ABB RobotStudio station: FinalProject.rsstnx

Station FinalProject (saved by RobotStudio 24.4.11080.0)
Controller IRB140_6_81
  mechanical unit ROB_1: IRB140_6_81_C_03, 6 joints, base frame (0, 0, 0) mm
Layout (positions relative to the parent item):
  - IRB140_6_81_C_03 [mechanism, from %ABB.RobotStudio.Models.IRB140%\IRB140_6_81_C_G_03.rslib] at (0, 0, 0) mm; joint values [0, 0, 0, 0, 0, 0] (rad or m)
  - VacuumGripper [mechanism] at (515, 0, 712) mm, rotated rx 0 ry 90 rz 0 deg
      TCP VacuumGripper at (122.78, 0, 0) mm, rotated rx 90 ry 45 rz 90 deg
      links: FakeEE
Attachment: VacuumGripper is attached to IRB140_6_81_C_03 / Link6
Targets, tools, work objects and paths stored in the station, written as RAPID:
! task T_ROB1
MODULE Numbers
  CONST robtarget T_01:=[[-310.742,318.894,0],[1,0,0,0],[0,0,0,0],[9E+09,9E+09,9E+09,9E+09,9E+09,9E+09]];
  CONST robtarget T_02:=[[-285.702,367.273,0],[1,0,0,0],[0,-1,0,0],[9E+09,9E+09,9E+09,9E+09,9E+09,9E+09]];
  CONST robtarget T_03:=[[-206.529,382.913,0],[1,0,0,0],[0,-1,0,0],[9E+09,9E+09,9E+09,9E+09,9E+09,9E+09]];
  CONST robtarget T_04:=[[-128.165,367.435,0],[1,0,0,0],[0,-2,1,0],[9E+09,9E+09,9E+09,9E+09,9E+09,9E+09]];
  CONST robtarget T_05:=[[-102.477,318.894,0],[1,0,0,0],[-2,0,1,6],[9E+09,9E+09,9E+09,9E+09,9E+09,9E+09]];
  CONST robtarget T_06:=[[-127.679,270.676,0],[1,0,0,0],[-2,0,1,6],[9E+09,9E+09,9E+09,9E+09,9E+09,9E+09]];
  CONST robtarget T_07:=[[-206.691,255.036,0],[1,0,0,0],[-1,0,-1,0],[9E+09,9E+09,9E+09,9E+09,9E+09,9E+09]];
  CONST robtarget T_08:=[[-284.811,270.514,0],[1,0,0,0],[-1,0,-1,0],[9E+09,9E+09,9E+09,9E+09,9E+09,9E+09]];
  CONST robtarget T_09:=[[-310.742,318.894,0],[1,0,0,0],[0,-1,0,0],[9E+09,9E+09,9E+09,9E+09,9E+09,9E+09]];
  CONST robtarget T_11:=[[-106.691,366.707,0],[1,0,0,0],[0,0,-1,1],[9E+09,9E+09,9E+09,9E+09,9E+09,9E+09]];
  CONST robtarget T_12:=[[-106.691,269.138,0],[1,0,0,0],[0,0,-1,1],[9E+09,9E+09,9E+09,9E+09,9E+09,9E+09]];
  CONST robtarget T_13:=[[-106.691,317.923,0],[1,0,0,0],[0,0,-1,1],[9E+09,9E+09,9E+09,9E+09,9E+09,9E+09]];
  CONST robtarget T_14:=[[-307.339,315.005,0],[1,0,0,0],[0,0,-1,1],[9E+09,9E+09,9E+09,9E+09,9E+09,9E+09]];
  CONST robtarget T_15:=[[-285.297,336.399,0],[1,0,0,0],[0,1,-2,1],[9E+09,9E+09,9E+09,9E+09,9E+09,9E+09]];
  CONST robtarget T_16:=[[-279.462,366.707,0],[1,0,0,0],[0,1,-2,1],[9E+09,9E+09,9E+09,9E+09,9E+09,9E+09]];
  CONST robtarget T_21:=[[-106.691,261.009,0],[1,0,0,0],[0,-1,0,0],[9E+09,9E+09,9E+09,9E+09,9E+09,9E+09]];
  CONST robtarget T_22:=[[-106.691,384.347,0],[1,0,0,0],[0,-2,1,0],[9E+09,9E+09,9E+09,9E+09,9E+09,9E+09]];
  CONST robtarget T_23:=[[-129.867,359.226,0],[1,0,0,0],[0,-2,1,0],[9E+09,9E+09,9E+09,9E+09,9E+09,9E+09]];
  CONST robtarget T_24:=[[-153.206,334.509,0],[1,0,0,0],[0,-2,1,0],[9E+09,9E+09,9E+09,9E+09,9E+09,9E+09]];
  CONST robtarget T_25:=[[-181.731,306.39,0],[1,0,0,0],[0,-1,0,0],[9E+09,9E+09,9E+09,9E+09,9E+09,9E+09]];
  CONST robtarget T_26:=[[-215.929,279.647,0],[1,0,0,0],[0,-1,0,0],[9E+09,9E+09,9E+09,9E+09,9E+09,9E+09]];
  CONST robtarget T_27:=[[-255.961,269.274,0],[1,0,0,0],[0,-1,0,0],[9E+09,9E+09,9E+09,9E+09,9E+09,9E+09]];
  CONST robtarget T_28:=[[-296.075,285.077,0],[1,0,0,0],[0,-1,0,0],[9E+09,9E+09,9E+09,9E+09,9E+09,9E+09]];
  CONST robtarget T_29:=[[-310.905,328.918,0],[1,0,0,0],[0,-1,0,0],[9E+09,9E+09,9E+09,9E+09,9E+09,9E+09]];
  CONST robtarget T_210:=[[-306.934,357.038,0],[1,0,0,0],[0,-1,0,0],[9E+09,9E+09,9E+09,9E+09,9E+09,9E+09]];
  CONST robtarget T_211:=[[-298.911,380.133,0],[1,0,0,0],[0,-1,0,0],[9E+09,9E+09,9E+09,9E+09,9E+09,9E+09]];
  CONST robtarget T_31:=[[-298.587,375.377,0],[1,0,0,0],[0,-1,0,0],[9E+09,9E+09,9E+09,9E+09,9E+09,9E+09]];
  CONST robtarget T_32:=[[-307.096,351.633,0],[1,0,0,0],[0,-1,0,0],[9E+09,9E+09,9E+09,9E+09,9E+09,9E+09]];
  CONST robtarget T_33:=[[-310.905,323.189,0],[1,0,0,0],[0,-1,0,0],[9E+09,9E+09,9E+09,9E+09,9E+09,9E+09]];
  CONST robtarget T_34:=[[-308.149,299.445,0],[1,0,0,0],[0,-1,0,0],[9E+09,9E+09,9E+09,9E+09,9E+09,9E+09]];
  CONST robtarget T_35:=[[-299.559,281.049,0],[1,0,0,0],[0,-1,0,0],[9E+09,9E+09,9E+09,9E+09,9E+09,9E+09]];
  CONST robtarget T_36:=[[-284.081,267.759,0],[1,0,0,0],[0,-1,0,0],[9E+09,9E+09,9E+09,9E+09,9E+09,9E+09]];
  CONST robtarget T_37:=[[-262.606,263.221,0],[1,0,0,0],[0,-1,0,0],[9E+09,9E+09,9E+09,9E+09,9E+09,9E+09]];
  CONST robtarget T_38:=[[-233.595,274.08,0],[1,0,0,0],[0,-1,0,0],[9E+09,9E+09,9E+09,9E+09,9E+09,9E+09]];
  CONST robtarget T_39:=[[-217.874,300.174,0],[1,0,0,0],[0,-1,0,0],[9E+09,9E+09,9E+09,9E+09,9E+09,9E+09]];
  CONST robtarget T_310:=[[-215.199,340.044,0],[1,0,0,0],[0,-1,0,0],[9E+09,9E+09,9E+09,9E+09,9E+09,9E+09]];
  CONST robtarget T_311:=[[-215.929,300.174,0],[1,0,0,0],[0,-1,0,0],[9E+09,9E+09,9E+09,9E+09,9E+09,9E+09]];
  CONST robtarget T_312:=[[-202.963,273.27,0],[1,0,0,0],[0,-1,0,0],[9E+09,9E+09,9E+09,9E+09,9E+09,9E+09]];
  CONST robtarget T_313:=[[-188.214,263.221,0],[1,0,0,0],[0,-1,0,0],[9E+09,9E+09,9E+09,9E+09,9E+09,9E+09]];
  CONST robtarget T_314:=[[-166.01,259.331,0],[1,0,0,0],[0,-1,0,0],[9E+09,9E+09,9E+09,9E+09,9E+09,9E+09]];
  CONST robtarget T_315:=[[-141.131,263.95,0],[1,0,0,0],[0,-1,0,0],[9E+09,9E+09,9E+09,9E+09,9E+09,9E+09]];
  CONST robtarget T_316:=[[-120.953,276.997,0],[1,0,0,0],[0,-1,0,0],[9E+09,9E+09,9E+09,9E+09,9E+09,9E+09]];
  CONST robtarget T_317:=[[-107.177,298.148,0],[1,0,0,0],[0,-2,1,0],[9E+09,9E+09,9E+09,9E+09,9E+09,9E+09]];
  CONST robtarget T_318:=[[-102.477,326.268,0],[1,0,0,0],[0,-2,1,0],[9E+09,9E+09,9E+09,9E+09,9E+09,9E+09]];
  CONST robtarget T_319:=[[-106.123,356.09,0],[1,0,0,0],[0,-2,1,0],[9E+09,9E+09,9E+09,9E+09,9E+09,9E+09]];
  CONST robtarget T_320:=[[-114.794,380.887,0],[1,0,0,0],[0,-2,1,0],[9E+09,9E+09,9E+09,9E+09,9E+09,9E+09]];
  CONST robtarget T_41:=[[-106.691,281.323,0],[1,0,0,0],[-1,-1,0,1],[9E+09,9E+09,9E+09,9E+09,9E+09,9E+09]];
  CONST robtarget T_42:=[[-306.691,281.323,0],[1,0,0,0],[0,0,-1,1],[9E+09,9E+09,9E+09,9E+09,9E+09,9E+09]];
  CONST robtarget T_43:=[[-306.691,305.958,0],[1,0,0,0],[0,1,-2,1],[9E+09,9E+09,9E+09,9E+09,9E+09,9E+09]];
  CONST robtarget T_44:=[[-203.611,395.424,0],[1,0,0,0],[0,1,-2,1],[9E+09,9E+09,9E+09,9E+09,9E+09,9E+09]];
  CONST robtarget T_45:=[[-175.41,395.424,0],[1,0,0,0],[0,1,-2,1],[9E+09,9E+09,9E+09,9E+09,9E+09,9E+09]];
  CONST robtarget T_46:=[[-175.41,257.498,0],[1,0,0,0],[0,1,-2,1],[9E+09,9E+09,9E+09,9E+09,9E+09,9E+09]];
  CONST robtarget T_51:=[[-306.691,269.007,0],[1,0,0,0],[0,1,-2,1],[9E+09,9E+09,9E+09,9E+09,9E+09,9E+09]];
  CONST robtarget T_52:=[[-306.691,378.732,0],[1,0,0,0],[0,1,-2,1],[9E+09,9E+09,9E+09,9E+09,9E+09,9E+09]];
  CONST robtarget T_53:=[[-223.611,378.732,0],[1,0,0,0],[0,1,-2,1],[9E+09,9E+09,9E+09,9E+09,9E+09,9E+09]];
  CONST robtarget T_54:=[[-229.867,352.962,0],[1,0,0,0],[0,1,-2,1],[9E+09,9E+09,9E+09,9E+09,9E+09,9E+09]];
  CONST robtarget T_55:=[[-231.002,334.809,0],[1,0,0,0],[0,1,-2,1],[9E+09,9E+09,9E+09,9E+09,9E+09,9E+09]];
  CONST robtarget T_56:=[[-228.49,308.796,0],[1,0,0,0],[0,1,-2,1],[9E+09,9E+09,9E+09,9E+09,9E+09,9E+09]];
  CONST robtarget T_57:=[[-218.522,288.456,0],[1,0,0,0],[0,1,-2,1],[9E+09,9E+09,9E+09,9E+09,9E+09,9E+09]];
  CONST robtarget T_58:=[[-199.721,273.221,0],[1,0,0,0],[0,1,-2,1],[9E+09,9E+09,9E+09,9E+09,9E+09,9E+09]];
  CONST robtarget T_59:=[[-170.224,267.873,0],[1,0,0,0],[0,1,-2,1],[9E+09,9E+09,9E+09,9E+09,9E+09,9E+09]];
  CONST robtarget T_510:=[[-143.482,272.492,0],[1,0,0,0],[0,0,-1,1],[9E+09,9E+09,9E+09,9E+09,9E+09,9E+09]];
  CONST robtarget T_511:=[[-122.088,285.539,0],[1,0,0,0],[0,0,-1,1],[9E+09,9E+09,9E+09,9E+09,9E+09,9E+09]];
  CONST robtarget T_512:=[[-107.744,306.527,0],[1,0,0,0],[0,0,-1,1],[9E+09,9E+09,9E+09,9E+09,9E+09,9E+09]];
  CONST robtarget T_513:=[[-102.477,334.647,0],[1,0,0,0],[0,0,-1,1],[9E+09,9E+09,9E+09,9E+09,9E+09,9E+09]];
  CONST robtarget T_514:=[[-105.637,362.848,0],[1,0,0,0],[0,0,-1,1],[9E+09,9E+09,9E+09,9E+09,9E+09,9E+09]];
  CONST robtarget T_515:=[[-113.822,386.997,0],[1,0,0,0],[0,0,-1,1],[9E+09,9E+09,9E+09,9E+09,9E+09,9E+09]];
  CONST robtarget T_61:=[[-307.663,280.947,0],[1,0,0,0],[0,0,-1,1],[9E+09,9E+09,9E+09,9E+09,9E+09,9E+09]];
  CONST robtarget T_62:=[[-310.418,303.638,0],[1,0,0,0],[0,1,-2,1],[9E+09,9E+09,9E+09,9E+09,9E+09,9E+09]];
  CONST robtarget T_63:=[[-301.909,343.346,0],[1,0,0,0],[0,1,-2,1],[9E+09,9E+09,9E+09,9E+09,9E+09,9E+09]];
  CONST robtarget T_64:=[[-278.165,371.385,0],[1,0,0,0],[0,1,-2,1],[9E+09,9E+09,9E+09,9E+09,9E+09,9E+09]];
  CONST robtarget T_65:=[[-241.618,387.916,0],[1,0,0,0],[0,1,-2,1],[9E+09,9E+09,9E+09,9E+09,9E+09,9E+09]];
  CONST robtarget T_66:=[[-194.535,393.265,0],[1,0,0,0],[0,1,-2,1],[9E+09,9E+09,9E+09,9E+09,9E+09,9E+09]];
  CONST robtarget T_67:=[[-149.721,387.43,0],[1,0,0,0],[0,1,-2,1],[9E+09,9E+09,9E+09,9E+09,9E+09,9E+09]];
  CONST robtarget T_68:=[[-120.629,371.223,0],[1,0,0,0],[0,0,-1,1],[9E+09,9E+09,9E+09,9E+09,9E+09,9E+09]];
  CONST robtarget T_69:=[[-107.015,351.693,0],[1,0,0,0],[0,0,-1,1],[9E+09,9E+09,9E+09,9E+09,9E+09,9E+09]];
  CONST robtarget T_610:=[[-102.477,327.138,0],[1,0,0,0],[0,0,-1,1],[9E+09,9E+09,9E+09,9E+09,9E+09,9E+09]];
  CONST robtarget T_611:=[[-107.258,302.503,0],[1,0,0,0],[0,0,-1,1],[9E+09,9E+09,9E+09,9E+09,9E+09,9E+09]];
  CONST robtarget T_612:=[[-121.277,282.406,0],[1,0,0,0],[0,0,-1,1],[9E+09,9E+09,9E+09,9E+09,9E+09,9E+09]];
  CONST robtarget T_613:=[[-143.076,268.71,0],[1,0,0,0],[0,0,-1,1],[9E+09,9E+09,9E+09,9E+09,9E+09,9E+09]];
  CONST robtarget T_614:=[[-171.52,263.605,0],[1,0,0,0],[0,1,-2,1],[9E+09,9E+09,9E+09,9E+09,9E+09,9E+09]];
  CONST robtarget T_615:=[[-201.504,268.954,0],[1,0,0,0],[0,1,-2,1],[9E+09,9E+09,9E+09,9E+09,9E+09,9E+09]];
  CONST robtarget T_616:=[[-222.574,285.323,0],[1,0,0,0],[0,1,-2,1],[9E+09,9E+09,9E+09,9E+09,9E+09,9E+09]];
  CONST robtarget T_617:=[[-232.055,303.638,0],[1,0,0,0],[0,1,-2,1],[9E+09,9E+09,9E+09,9E+09,9E+09,9E+09]];
  CONST robtarget T_618:=[[-234.405,324.059,0],[1,0,0,0],[0,1,-2,1],[9E+09,9E+09,9E+09,9E+09,9E+09,9E+09]];
  CONST robtarget T_619:=[[-230.759,346.101,0],[1,0,0,0],[0,1,-2,1],[9E+09,9E+09,9E+09,9E+09,9E+09,9E+09]];
  CONST robtarget T_620:=[[-220.467,365.712,0],[1,0,0,0],[0,1,-2,1],[9E+09,9E+09,9E+09,9E+09,9E+09,9E+09]];
  CONST robtarget T_621:=[[-194.535,393.265,0],[1,0,0,0],[0,1,-2,1],[9E+09,9E+09,9E+09,9E+09,9E+09,9E+09]];
  CONST robtarget T_71:=[[-306.691,388.239,0],[1,0,0,0],[0,-1,0,0],[9E+09,9E+09,9E+09,9E+09,9E+09,9E+09]];
  CONST robtarget T_72:=[[-306.691,261.334,0],[1,0,0,0],[0,-1,0,0],[9E+09,9E+09,9E+09,9E+09,9E+09,9E+09]];
  CONST robtarget T_73:=[[-106.691,347.882,0],[1,0,0,0],[0,-1,0,0],[9E+09,9E+09,9E+09,9E+09,9E+09,9E+09]];
  CONST robtarget T_81:=[[-214.308,359.688,0],[1,0,0,0],[0,1,-2,1],[9E+09,9E+09,9E+09,9E+09,9E+09,9E+09]];
  CONST robtarget T_82:=[[-233.109,381.568,0],[1,0,0,0],[0,1,-2,1],[9E+09,9E+09,9E+09,9E+09,9E+09,9E+09]];
  CONST robtarget T_83:=[[-258.554,388.699,0],[1,0,0,0],[0,1,-2,1],[9E+09,9E+09,9E+09,9E+09,9E+09,9E+09]];
  CONST robtarget T_84:=[[-296.156,371.681,0],[1,0,0,0],[0,1,-2,1],[9E+09,9E+09,9E+09,9E+09,9E+09,9E+09]];
  CONST robtarget T_85:=[[-311.229,328.407,0],[1,0,0,0],[0,1,-2,1],[9E+09,9E+09,9E+09,9E+09,9E+09,9E+09]];
  CONST robtarget T_86:=[[-296.966,284.728,0],[1,0,0,0],[0,1,-2,1],[9E+09,9E+09,9E+09,9E+09,9E+09,9E+09]];
  CONST robtarget T_87:=[[-260.337,268.278,0],[1,0,0,0],[0,1,-2,1],[9E+09,9E+09,9E+09,9E+09,9E+09,9E+09]];
  CONST robtarget T_88:=[[-233.757,276.138,0],[1,0,0,0],[0,1,-2,1],[9E+09,9E+09,9E+09,9E+09,9E+09,9E+09]];
  CONST robtarget T_89:=[[-213.174,298.748,0],[1,0,0,0],[0,1,-2,1],[9E+09,9E+09,9E+09,9E+09,9E+09,9E+09]];
  CONST robtarget T_810:=[[-213.498,359.688,0],[1,0,0,0],[0,1,-2,1],[9E+09,9E+09,9E+09,9E+09,9E+09,9E+09]];
  CONST robtarget T_811:=[[-191.78,384.89,0],[1,0,0,0],[0,1,-2,1],[9E+09,9E+09,9E+09,9E+09,9E+09,9E+09]];
  CONST robtarget T_812:=[[-161.958,393.561,0],[1,0,0,0],[0,1,-2,1],[9E+09,9E+09,9E+09,9E+09,9E+09,9E+09]];
  CONST robtarget T_813:=[[-138.457,389.185,0],[1,0,0,0],[0,0,-1,1],[9E+09,9E+09,9E+09,9E+09,9E+09,9E+09]];
  CONST robtarget T_814:=[[-119.332,376.381,0],[1,0,0,0],[0,0,-1,1],[9E+09,9E+09,9E+09,9E+09,9E+09,9E+09]];
  CONST robtarget T_815:=[[-106.61,355.555,0],[1,0,0,0],[0,0,-1,1],[9E+09,9E+09,9E+09,9E+09,9E+09,9E+09]];
  CONST robtarget T_816:=[[-102.152,328.407,0],[1,0,0,0],[0,0,-1,1],[9E+09,9E+09,9E+09,9E+09,9E+09,9E+09]];
  CONST robtarget T_817:=[[-119.494,281.892,0],[1,0,0,0],[0,0,-1,1],[9E+09,9E+09,9E+09,9E+09,9E+09,9E+09]];
  CONST robtarget T_818:=[[-162.444,263.253,0],[1,0,0,0],[0,1,-2,1],[9E+09,9E+09,9E+09,9E+09,9E+09,9E+09]];
  CONST robtarget T_819:=[[-192.59,272.249,0],[1,0,0,0],[0,1,-2,1],[9E+09,9E+09,9E+09,9E+09,9E+09,9E+09]];
  CONST robtarget T_820:=[[-212.363,298.748,0],[1,0,0,0],[0,1,-2,1],[9E+09,9E+09,9E+09,9E+09,9E+09,9E+09]];
  CONST robtarget T_821:=[[-214.308,359.688,0],[1,0,0,0],[0,1,-2,1],[9E+09,9E+09,9E+09,9E+09,9E+09,9E+09]];
  CONST robtarget T_91:=[[-105.556,371.949,0],[1,0,0,0],[0,0,-1,1],[9E+09,9E+09,9E+09,9E+09,9E+09,9E+09]];
  CONST robtarget T_92:=[[-102.801,349.258,0],[1,0,0,0],[0,0,-1,1],[9E+09,9E+09,9E+09,9E+09,9E+09,9E+09]];
  CONST robtarget T_93:=[[-110.986,309.388,0],[1,0,0,0],[0,0,-1,1],[9E+09,9E+09,9E+09,9E+09,9E+09,9E+09]];
  CONST robtarget T_94:=[[-134.729,281.673,0],[1,0,0,0],[0,0,-1,1],[9E+09,9E+09,9E+09,9E+09,9E+09,9E+09]];
  CONST robtarget T_95:=[[-171.682,265.223,0],[1,0,0,0],[0,1,-2,1],[9E+09,9E+09,9E+09,9E+09,9E+09,9E+09]];
  CONST robtarget T_96:=[[-218.684,259.631,0],[1,0,0,0],[0,1,-2,1],[9E+09,9E+09,9E+09,9E+09,9E+09,9E+09]];
  CONST robtarget T_97:=[[-263.903,265.304,0],[1,0,0,0],[0,1,-2,1],[9E+09,9E+09,9E+09,9E+09,9E+09,9E+09]];
  CONST robtarget T_98:=[[-292.752,281.349,0],[1,0,0,0],[0,1,-2,1],[9E+09,9E+09,9E+09,9E+09,9E+09,9E+09]];
  CONST robtarget T_99:=[[-306.123,300.798,0],[1,0,0,0],[0,1,-2,1],[9E+09,9E+09,9E+09,9E+09,9E+09,9E+09]];
  CONST robtarget T_910:=[[-310.742,325.757,0],[1,0,0,0],[0,1,-2,1],[9E+09,9E+09,9E+09,9E+09,9E+09,9E+09]];
  CONST robtarget T_911:=[[-305.799,350.15,0],[1,0,0,0],[0,1,-2,1],[9E+09,9E+09,9E+09,9E+09,9E+09,9E+09]];
  CONST robtarget T_912:=[[-291.942,370.49,0],[1,0,0,0],[0,1,-2,1],[9E+09,9E+09,9E+09,9E+09,9E+09,9E+09]];
  CONST robtarget T_913:=[[-269.9,384.266,0],[1,0,0,0],[0,1,-2,1],[9E+09,9E+09,9E+09,9E+09,9E+09,9E+09]];
  CONST robtarget T_914:=[[-241.699,389.291,0],[1,0,0,0],[0,1,-2,1],[9E+09,9E+09,9E+09,9E+09,9E+09,9E+09]];
  CONST robtarget T_915:=[[-211.472,383.78,0],[1,0,0,0],[0,1,-2,1],[9E+09,9E+09,9E+09,9E+09,9E+09,9E+09]];
  CONST robtarget T_916:=[[-190.645,367.573,0],[1,0,0,0],[0,1,-2,1],[9E+09,9E+09,9E+09,9E+09,9E+09,9E+09]];
  CONST robtarget T_917:=[[-181.245,349.177,0],[1,0,0,0],[0,1,-2,1],[9E+09,9E+09,9E+09,9E+09,9E+09,9E+09]];
  CONST robtarget T_918:=[[-178.814,328.999,0],[1,0,0,0],[0,1,-2,1],[9E+09,9E+09,9E+09,9E+09,9E+09,9E+09]];
  CONST robtarget T_919:=[[-182.136,307.767,0],[1,0,0,0],[0,1,-2,1],[9E+09,9E+09,9E+09,9E+09,9E+09,9E+09]];
  CONST robtarget T_920:=[[-192.752,287.346,0],[1,0,0,0],[0,1,-2,1],[9E+09,9E+09,9E+09,9E+09,9E+09,9E+09]];
  CONST robtarget T_921:=[[-218.684,259.631,0],[1,0,0,0],[0,1,-2,1],[9E+09,9E+09,9E+09,9E+09,9E+09,9E+09]];
  CONST robtarget T_921_2:=[[-218.684,259.631,0],[1,0,0,0],[-1,-2,1,1],[9E+09,9E+09,9E+09,9E+09,9E+09,9E+09]];
  CONST robtarget T_01_2:=[[-310.742,318.894,0],[1,0,0,0],[0,0,0,0],[9E+09,9E+09,9E+09,9E+09,9E+09,9E+09]];
  CONST robtarget T_02_2:=[[-285.702,367.273,0],[1,0,0,0],[-1,0,-1,0],[9E+09,9E+09,9E+09,9E+09,9E+09,9E+09]];
  CONST robtarget T_03_2:=[[-206.529,382.913,0],[1,0,0,0],[-1,0,-1,0],[9E+09,9E+09,9E+09,9E+09,9E+09,9E+09]];
  CONST robtarget T_04_2:=[[-128.165,367.435,0],[1,0,0,0],[-1,0,-1,0],[9E+09,9E+09,9E+09,9E+09,9E+09,9E+09]];
  CONST robtarget T_05_2:=[[-102.477,318.894,0],[1,0,0,0],[-1,0,-1,0],[9E+09,9E+09,9E+09,9E+09,9E+09,9E+09]];
  CONST robtarget T_06_2:=[[-127.679,270.676,0],[1,0,0,0],[-1,1,-2,0],[9E+09,9E+09,9E+09,9E+09,9E+09,9E+09]];
  CONST robtarget T_07_2:=[[-206.691,255.036,0],[1,0,0,0],[-1,0,-1,0],[9E+09,9E+09,9E+09,9E+09,9E+09,9E+09]];
  CONST robtarget T_08_2:=[[-284.811,270.514,0],[1,0,0,0],[-1,0,-1,0],[9E+09,9E+09,9E+09,9E+09,9E+09,9E+09]];
  CONST robtarget T_09_2:=[[-310.742,318.894,0],[1,0,0,0],[-1,0,-1,0],[9E+09,9E+09,9E+09,9E+09,9E+09,9E+09]];
  CONST robtarget T_11_2:=[[-106.691,366.707,0],[1,0,0,0],[-1,1,-2,0],[9E+09,9E+09,9E+09,9E+09,9E+09,9E+09]];
  CONST robtarget T_12_2:=[[-106.691,269.138,0],[1,0,0,0],[-1,1,-2,0],[9E+09,9E+09,9E+09,9E+09,9E+09,9E+09]];
  CONST robtarget T_13_2:=[[-106.691,317.923,0],[1,0,0,0],[-1,1,-2,0],[9E+09,9E+09,9E+09,9E+09,9E+09,9E+09]];
  CONST robtarget T_14_2:=[[-307.339,315.005,0],[1,0,0,0],[-1,1,-2,0],[9E+09,9E+09,9E+09,9E+09,9E+09,9E+09]];
  CONST robtarget T_15_2:=[[-285.297,336.399,0],[1,0,0,0],[-1,0,-1,0],[9E+09,9E+09,9E+09,9E+09,9E+09,9E+09]];
  CONST robtarget T_16_2:=[[-279.462,366.707,0],[1,0,0,0],[-1,0,-1,0],[9E+09,9E+09,9E+09,9E+09,9E+09,9E+09]];
  CONST robtarget T_21_2:=[[-106.691,261.009,0],[1,0,0,0],[-1,1,-2,0],[9E+09,9E+09,9E+09,9E+09,9E+09,9E+09]];
  CONST robtarget T_22_2:=[[-106.691,384.347,0],[1,0,0,0],[-1,1,-2,0],[9E+09,9E+09,9E+09,9E+09,9E+09,9E+09]];
  CONST robtarget T_23_2:=[[-129.867,359.226,0],[1,0,0,0],[-1,1,-2,0],[9E+09,9E+09,9E+09,9E+09,9E+09,9E+09]];
  CONST robtarget T_24_2:=[[-153.206,334.509,0],[1,0,0,0],[-1,0,-1,0],[9E+09,9E+09,9E+09,9E+09,9E+09,9E+09]];
  CONST robtarget T_25_2:=[[-181.731,306.39,0],[1,0,0,0],[-1,0,-1,0],[9E+09,9E+09,9E+09,9E+09,9E+09,9E+09]];
  CONST robtarget T_26_2:=[[-215.929,279.647,0],[1,0,0,0],[-1,0,-1,0],[9E+09,9E+09,9E+09,9E+09,9E+09,9E+09]];
  CONST robtarget T_27_2:=[[-255.961,269.274,0],[1,0,0,0],[-1,0,-1,0],[9E+09,9E+09,9E+09,9E+09,9E+09,9E+09]];
  CONST robtarget T_28_2:=[[-296.075,285.077,0],[1,0,0,0],[-1,0,-1,0],[9E+09,9E+09,9E+09,9E+09,9E+09,9E+09]];
  CONST robtarget T_29_2:=[[-310.905,328.918,0],[1,0,0,0],[-1,0,-1,0],[9E+09,9E+09,9E+09,9E+09,9E+09,9E+09]];
  CONST robtarget T_210_2:=[[-306.934,357.038,0],[1,0,0,0],[-1,0,-1,0],[9E+09,9E+09,9E+09,9E+09,9E+09,9E+09]];
  CONST robtarget T_211_2:=[[-298.911,380.133,0],[1,0,0,0],[-1,0,-1,0],[9E+09,9E+09,9E+09,9E+09,9E+09,9E+09]];
  CONST robtarget T_31_2:=[[-298.587,375.377,0],[1,0,0,0],[0,-1,0,0],[9E+09,9E+09,9E+09,9E+09,9E+09,9E+09]];
  CONST robtarget T_32_2:=[[-307.096,351.633,0],[1,0,0,0],[-1,0,-1,0],[9E+09,9E+09,9E+09,9E+09,9E+09,9E+09]];
  CONST robtarget T_33_2:=[[-310.905,323.189,0],[1,0,0,0],[-1,0,-1,0],[9E+09,9E+09,9E+09,9E+09,9E+09,9E+09]];
  CONST robtarget T_34_2:=[[-308.149,299.445,0],[1,0,0,0],[-1,0,-1,0],[9E+09,9E+09,9E+09,9E+09,9E+09,9E+09]];
  CONST robtarget T_35_2:=[[-299.559,281.049,0],[1,0,0,0],[-1,0,-1,0],[9E+09,9E+09,9E+09,9E+09,9E+09,9E+09]];
  CONST robtarget T_36_2:=[[-284.081,267.759,0],[1,0,0,0],[-1,0,-1,0],[9E+09,9E+09,9E+09,9E+09,9E+09,9E+09]];
  CONST robtarget T_37_2:=[[-262.606,263.221,0],[1,0,0,0],[-1,0,-1,0],[9E+09,9E+09,9E+09,9E+09,9E+09,9E+09]];
  CONST robtarget T_38_2:=[[-233.595,274.08,0],[1,0,0,0],[-1,0,-1,0],[9E+09,9E+09,9E+09,9E+09,9E+09,9E+09]];
  CONST robtarget T_39_2:=[[-217.874,300.174,0],[1,0,0,0],[-1,0,-1,0],[9E+09,9E+09,9E+09,9E+09,9E+09,9E+09]];
  CONST robtarget T_310_2:=[[-215.199,340.044,0],[1,0,0,0],[0,-1,0,0],[9E+09,9E+09,9E+09,9E+09,9E+09,9E+09]];
  CONST robtarget T_311_2:=[[-215.929,300.174,0],[1,0,0,0],[0,-1,0,0],[9E+09,9E+09,9E+09,9E+09,9E+09,9E+09]];
  CONST robtarget T_312_2:=[[-202.963,273.27,0],[1,0,0,0],[0,-1,0,0],[9E+09,9E+09,9E+09,9E+09,9E+09,9E+09]];
  CONST robtarget T_313_2:=[[-188.214,263.221,0],[1,0,0,0],[0,-1,0,0],[9E+09,9E+09,9E+09,9E+09,9E+09,9E+09]];
  CONST robtarget T_314_2:=[[-166.01,259.331,0],[1,0,0,0],[0,-1,0,0],[9E+09,9E+09,9E+09,9E+09,9E+09,9E+09]];
  CONST robtarget T_315_2:=[[-141.131,263.95,0],[1,0,0,0],[0,-1,0,0],[9E+09,9E+09,9E+09,9E+09,9E+09,9E+09]];
  CONST robtarget T_316_2:=[[-120.953,276.997,0],[1,0,0,0],[-1,1,-2,0],[9E+09,9E+09,9E+09,9E+09,9E+09,9E+09]];
  CONST robtarget T_317_2:=[[-107.177,298.148,0],[1,0,0,0],[-1,1,-2,0],[9E+09,9E+09,9E+09,9E+09,9E+09,9E+09]];
  CONST robtarget T_318_2:=[[-102.477,326.268,0],[1,0,0,0],[-1,1,-2,0],[9E+09,9E+09,9E+09,9E+09,9E+09,9E+09]];
  CONST robtarget T_319_2:=[[-106.123,356.09,0],[1,0,0,0],[-1,1,-2,0],[9E+09,9E+09,9E+09,9E+09,9E+09,9E+09]];
  CONST robtarget T_320_2:=[[-114.794,380.887,0],[1,0,0,0],[0,-2,1,0],[9E+09,9E+09,9E+09,9E+09,9E+09,9E+09]];
  CONST robtarget T_41_2:=[[-106.691,281.323,0],[1,0,0,0],[-1,1,-2,0],[9E+09,9E+09,9E+09,9E+09,9E+09,9E+09]];
  CONST robtarget T_42_2:=[[-306.691,281.323,0],[1,0,0,0],[-1,0,-1,0],[9E+09,9E+09,9E+09,9E+09,9E+09,9E+09]];
  CONST robtarget T_43_2:=[[-306.691,305.958,0],[1,0,0,0],[-1,0,-1,0],[9E+09,9E+09,9E+09,9E+09,9E+09,9E+09]];
  CONST robtarget T_44_2:=[[-203.611,395.424,0],[1,0,0,0],[0,-1,0,0],[9E+09,9E+09,9E+09,9E+09,9E+09,9E+09]];
  CONST robtarget T_45_2:=[[-175.41,395.424,0],[1,0,0,0],[0,-1,0,0],[9E+09,9E+09,9E+09,9E+09,9E+09,9E+09]];
  CONST robtarget T_46_2:=[[-175.41,257.498,0],[1,0,0,0],[-1,0,-1,0],[9E+09,9E+09,9E+09,9E+09,9E+09,9E+09]];
  CONST robtarget T_51_2:=[[-306.691,269.007,0],[1,0,0,0],[-1,0,-1,0],[9E+09,9E+09,9E+09,9E+09,9E+09,9E+09]];
  CONST robtarget T_52_2:=[[-306.691,378.732,0],[1,0,0,0],[0,-1,0,0],[9E+09,9E+09,9E+09,9E+09,9E+09,9E+09]];
  CONST robtarget T_53_2:=[[-223.611,378.732,0],[1,0,0,0],[0,-1,0,0],[9E+09,9E+09,9E+09,9E+09,9E+09,9E+09]];
  CONST robtarget T_54_2:=[[-229.867,352.962,0],[1,0,0,0],[-1,0,-1,0],[9E+09,9E+09,9E+09,9E+09,9E+09,9E+09]];
  CONST robtarget T_55_2:=[[-231.002,334.809,0],[1,0,0,0],[-1,0,-1,0],[9E+09,9E+09,9E+09,9E+09,9E+09,9E+09]];
  CONST robtarget T_56_2:=[[-228.49,308.796,0],[1,0,0,0],[-1,0,-1,0],[9E+09,9E+09,9E+09,9E+09,9E+09,9E+09]];
  CONST robtarget T_57_2:=[[-218.522,288.456,0],[1,0,0,0],[-1,0,-1,0],[9E+09,9E+09,9E+09,9E+09,9E+09,9E+09]];
  CONST robtarget T_58_2:=[[-199.721,273.221,0],[1,0,0,0],[-1,0,-1,0],[9E+09,9E+09,9E+09,9E+09,9E+09,9E+09]];
  CONST robtarget T_59_2:=[[-170.224,267.873,0],[1,0,0,0],[-1,0,-1,0],[9E+09,9E+09,9E+09,9E+09,9E+09,9E+09]];
  CONST robtarget T_510_2:=[[-143.482,272.492,0],[1,0,0,0],[-1,0,-1,0],[9E+09,9E+09,9E+09,9E+09,9E+09,9E+09]];
  CONST robtarget T_511_2:=[[-122.088,285.539,0],[1,0,0,0],[0,0,-1,1],[9E+09,9E+09,9E+09,9E+09,9E+09,9E+09]];
  CONST robtarget T_512_2:=[[-107.744,306.527,0],[1,0,0,0],[0,0,-1,1],[9E+09,9E+09,9E+09,9E+09,9E+09,9E+09]];
  CONST robtarget T_513_2:=[[-102.477,334.647,0],[1,0,0,0],[0,0,-1,1],[9E+09,9E+09,9E+09,9E+09,9E+09,9E+09]];
  CONST robtarget T_514_2:=[[-105.637,362.848,0],[1,0,0,0],[0,0,-1,1],[9E+09,9E+09,9E+09,9E+09,9E+09,9E+09]];
  CONST robtarget T_515_2:=[[-113.822,386.997,0],[1,0,0,0],[0,0,-1,1],[9E+09,9E+09,9E+09,9E+09,9E+09,9E+09]];
  CONST robtarget T_61_2:=[[-307.663,280.947,0],[1,0,0,0],[-1,0,-1,0],[9E+09,9E+09,9E+09,9E+09,9E+09,9E+09]];
  CONST robtarget T_62_2:=[[-310.418,303.638,0],[1,0,0,0],[-1,0,-1,0],[9E+09,9E+09,9E+09,9E+09,9E+09,9E+09]];
  CONST robtarget T_63_2:=[[-301.909,343.346,0],[1,0,0,0],[-1,0,-1,0],[9E+09,9E+09,9E+09,9E+09,9E+09,9E+09]];
  CONST robtarget T_64_2:=[[-278.165,371.385,0],[1,0,0,0],[0,-1,0,0],[9E+09,9E+09,9E+09,9E+09,9E+09,9E+09]];
  CONST robtarget T_65_2:=[[-241.618,387.916,0],[1,0,0,0],[0,-1,0,0],[9E+09,9E+09,9E+09,9E+09,9E+09,9E+09]];
  CONST robtarget T_66_2:=[[-194.535,393.265,0],[1,0,0,0],[0,-1,0,0],[9E+09,9E+09,9E+09,9E+09,9E+09,9E+09]];
  CONST robtarget T_67_2:=[[-149.721,387.43,0],[1,0,0,0],[0,-1,0,0],[9E+09,9E+09,9E+09,9E+09,9E+09,9E+09]];
  CONST robtarget T_68_2:=[[-120.629,371.223,0],[1,0,0,0],[0,-1,0,0],[9E+09,9E+09,9E+09,9E+09,9E+09,9E+09]];
  CONST robtarget T_69_2:=[[-107.015,351.693,0],[1,0,0,0],[-1,1,-2,0],[9E+09,9E+09,9E+09,9E+09,9E+09,9E+09]];
  CONST robtarget T_610_2:=[[-102.477,327.138,0],[1,0,0,0],[0,0,-1,1],[9E+09,9E+09,9E+09,9E+09,9E+09,9E+09]];
  CONST robtarget T_611_2:=[[-107.258,302.503,0],[1,0,0,0],[0,0,-1,1],[9E+09,9E+09,9E+09,9E+09,9E+09,9E+09]];
  CONST robtarget T_612_2:=[[-121.277,282.406,0],[1,0,0,0],[0,0,-1,1],[9E+09,9E+09,9E+09,9E+09,9E+09,9E+09]];
  CONST robtarget T_613_2:=[[-143.076,268.71,0],[1,0,0,0],[-1,-2,1,1],[9E+09,9E+09,9E+09,9E+09,9E+09,9E+09]];
  CONST robtarget T_614_2:=[[-171.52,263.605,0],[1,0,0,0],[-1,-2,1,1],[9E+09,9E+09,9E+09,9E+09,9E+09,9E+09]];
  CONST robtarget T_615_2:=[[-201.504,268.954,0],[1,0,0,0],[-1,-2,1,1],[9E+09,9E+09,9E+09,9E+09,9E+09,9E+09]];
  CONST robtarget T_616_2:=[[-222.574,285.323,0],[1,0,0,0],[-1,-2,1,1],[9E+09,9E+09,9E+09,9E+09,9E+09,9E+09]];
  CONST robtarget T_617_2:=[[-232.055,303.638,0],[1,0,0,0],[-1,-2,1,1],[9E+09,9E+09,9E+09,9E+09,9E+09,9E+09]];
  CONST robtarget T_618_2:=[[-234.405,324.059,0],[1,0,0,0],[-1,-2,1,1],[9E+09,9E+09,9E+09,9E+09,9E+09,9E+09]];
  CONST robtarget T_619_2:=[[-230.759,346.101,0],[1,0,0,0],[-1,-2,1,1],[9E+09,9E+09,9E+09,9E+09,9E+09,9E+09]];
  CONST robtarget T_620_2:=[[-220.467,365.712,0],[1,0,0,0],[0,1,-2,1],[9E+09,9E+09,9E+09,9E+09,9E+09,9E+09]];
  CONST robtarget T_621_2:=[[-194.535,393.265,0],[1,0,0,0],[0,1,-2,1],[9E+09,9E+09,9E+09,9E+09,9E+09,9E+09]];
  CONST robtarget T_71_2:=[[-306.691,388.239,0],[1,0,0,0],[0,-1,0,0],[9E+09,9E+09,9E+09,9E+09,9E+09,9E+09]];
  CONST robtarget T_72_2:=[[-306.691,261.334,0],[1,0,0,0],[-1,0,-1,0],[9E+09,9E+09,9E+09,9E+09,9E+09,9E+09]];
  CONST robtarget T_73_2:=[[-106.691,347.882,0],[1,0,0,0],[-1,1,-2,0],[9E+09,9E+09,9E+09,9E+09,9E+09,9E+09]];
  CONST robtarget T_81_2:=[[-214.308,359.688,0],[1,0,0,0],[-1,0,-1,0],[9E+09,9E+09,9E+09,9E+09,9E+09,9E+09]];
  CONST robtarget T_82_2:=[[-233.109,381.568,0],[1,0,0,0],[0,-1,0,0],[9E+09,9E+09,9E+09,9E+09,9E+09,9E+09]];
  CONST robtarget T_83_2:=[[-258.554,388.699,0],[1,0,0,0],[0,-1,0,0],[9E+09,9E+09,9E+09,9E+09,9E+09,9E+09]];
  CONST robtarget T_84_2:=[[-296.156,371.681,0],[1,0,0,0],[0,-1,0,0],[9E+09,9E+09,9E+09,9E+09,9E+09,9E+09]];
  CONST robtarget T_85_2:=[[-311.229,328.407,0],[1,0,0,0],[-1,0,-1,0],[9E+09,9E+09,9E+09,9E+09,9E+09,9E+09]];
  CONST robtarget T_86_2:=[[-296.966,284.728,0],[1,0,0,0],[-1,0,-1,0],[9E+09,9E+09,9E+09,9E+09,9E+09,9E+09]];
  CONST robtarget T_87_2:=[[-260.337,268.278,0],[1,0,0,0],[-1,0,-1,0],[9E+09,9E+09,9E+09,9E+09,9E+09,9E+09]];
  CONST robtarget T_88_2:=[[-233.757,276.138,0],[1,0,0,0],[-1,0,-1,0],[9E+09,9E+09,9E+09,9E+09,9E+09,9E+09]];
  CONST robtarget T_89_2:=[[-213.174,298.748,0],[1,0,0,0],[-1,0,-1,0],[9E+09,9E+09,9E+09,9E+09,9E+09,9E+09]];
  CONST robtarget T_810_2:=[[-213.498,359.688,0],[1,0,0,0],[0,1,-2,1],[9E+09,9E+09,9E+09,9E+09,9E+09,9E+09]];
  CONST robtarget T_811_2:=[[-191.78,384.89,0],[1,0,0,0],[0,1,-2,1],[9E+09,9E+09,9E+09,9E+09,9E+09,9E+09]];
  CONST robtarget T_812_2:=[[-161.958,393.561,0],[1,0,0,0],[0,1,-2,1],[9E+09,9E+09,9E+09,9E+09,9E+09,9E+09]];
  CONST robtarget T_813_2:=[[-138.457,389.185,0],[1,0,0,0],[0,0,-1,1],[9E+09,9E+09,9E+09,9E+09,9E+09,9E+09]];
  CONST robtarget T_814_2:=[[-119.332,376.381,0],[1,0,0,0],[0,0,-1,1],[9E+09,9E+09,9E+09,9E+09,9E+09,9E+09]];
  CONST robtarget T_815_2:=[[-106.61,355.555,0],[1,0,0,0],[0,0,-1,1],[9E+09,9E+09,9E+09,9E+09,9E+09,9E+09]];
  CONST robtarget T_816_2:=[[-102.152,328.407,0],[1,0,0,0],[0,0,-1,1],[9E+09,9E+09,9E+09,9E+09,9E+09,9E+09]];
  CONST robtarget T_817_2:=[[-119.494,281.892,0],[1,0,0,0],[0,0,-1,1],[9E+09,9E+09,9E+09,9E+09,9E+09,9E+09]];
  CONST robtarget T_818_2:=[[-162.444,263.253,0],[1,0,0,0],[-1,-2,1,1],[9E+09,9E+09,9E+09,9E+09,9E+09,9E+09]];
  CONST robtarget T_819_2:=[[-192.59,272.249,0],[1,0,0,0],[-1,-2,1,1],[9E+09,9E+09,9E+09,9E+09,9E+09,9E+09]];
  CONST robtarget T_820_2:=[[-212.363,298.748,0],[1,0,0,0],[-1,-2,1,1],[9E+09,9E+09,9E+09,9E+09,9E+09,9E+09]];
  CONST robtarget T_821_2:=[[-214.308,359.688,0],[1,0,0,0],[0,1,-2,1],[9E+09,9E+09,9E+09,9E+09,9E+09,9E+09]];
  CONST robtarget T_91_2:=[[-105.556,371.949,0],[1,0,0,0],[0,0,-1,1],[9E+09,9E+09,9E+09,9E+09,9E+09,9E+09]];
  CONST robtarget T_92_2:=[[-102.801,349.258,0],[1,0,0,0],[0,0,-1,1],[9E+09,9E+09,9E+09,9E+09,9E+09,9E+09]];
  CONST robtarget T_93_2:=[[-110.986,309.388,0],[1,0,0,0],[0,0,-1,1],[9E+09,9E+09,9E+09,9E+09,9E+09,9E+09]];
  CONST robtarget T_94_2:=[[-134.729,281.673,0],[1,0,0,0],[-1,-2,1,1],[9E+09,9E+09,9E+09,9E+09,9E+09,9E+09]];
  CONST robtarget T_95_2:=[[-171.682,265.223,0],[1,0,0,0],[-1,-2,1,1],[9E+09,9E+09,9E+09,9E+09,9E+09,9E+09]];
  CONST robtarget T_96_2:=[[-218.684,259.631,0],[1,0,0,0],[-1,-2,1,1],[9E+09,9E+09,9E+09,9E+09,9E+09,9E+09]];
  CONST robtarget T_97_2:=[[-263.903,265.304,0],[1,0,0,0],[-1,-2,1,1],[9E+09,9E+09,9E+09,9E+09,9E+09,9E+09]];
  CONST robtarget T_98_2:=[[-292.752,281.349,0],[1,0,0,0],[-1,-2,1,1],[9E+09,9E+09,9E+09,9E+09,9E+09,9E+09]];
  CONST robtarget T_99_2:=[[-306.123,300.798,0],[1,0,0,0],[-1,-2,1,1],[9E+09,9E+09,9E+09,9E+09,9E+09,9E+09]];
  CONST robtarget T_910_2:=[[-310.742,325.757,0],[1,0,0,0],[-1,-2,1,1],[9E+09,9E+09,9E+09,9E+09,9E+09,9E+09]];
  CONST robtarget T_911_2:=[[-305.799,350.15,0],[1,0,0,0],[0,1,-2,1],[9E+09,9E+09,9E+09,9E+09,9E+09,9E+09]];
  CONST robtarget T_912_2:=[[-291.942,370.49,0],[1,0,0,0],[0,1,-2,1],[9E+09,9E+09,9E+09,9E+09,9E+09,9E+09]];
  CONST robtarget T_913_2:=[[-269.9,384.266,0],[1,0,0,0],[0,1,-2,1],[9E+09,9E+09,9E+09,9E+09,9E+09,9E+09]];
  CONST robtarget T_914_2:=[[-241.699,389.291,0],[1,0,0,0],[0,1,-2,1],[9E+09,9E+09,9E+09,9E+09,9E+09,9E+09]];
  CONST robtarget T_915_2:=[[-211.472,383.78,0],[1,0,0,0],[0,1,-2,1],[9E+09,9E+09,9E+09,9E+09,9E+09,9E+09]];
  CONST robtarget T_916_2:=[[-190.645,367.573,0],[1,0,0,0],[0,1,-2,1],[9E+09,9E+09,9E+09,9E+09,9E+09,9E+09]];
  CONST robtarget T_917_2:=[[-181.245,349.177,0],[1,0,0,0],[-1,-2,1,1],[9E+09,9E+09,9E+09,9E+09,9E+09,9E+09]];
  CONST robtarget T_918_2:=[[-178.814,328.999,0],[1,0,0,0],[-1,-2,1,1],[9E+09,9E+09,9E+09,9E+09,9E+09,9E+09]];
  CONST robtarget T_919_2:=[[-182.136,307.767,0],[1,0,0,0],[-1,-2,1,1],[9E+09,9E+09,9E+09,9E+09,9E+09,9E+09]];
  CONST robtarget T_920_2:=[[-192.752,287.346,0],[1,0,0,0],[-1,-2,1,1],[9E+09,9E+09,9E+09,9E+09,9E+09,9E+09]];
ENDMODULE

! task T_ROB1
MODULE MainModule
  PERS tooldata VacuumGripper:=[TRUE,[[0,0,129.78],[1,0,0,0]],[1,[0,0,1],[1,0,0,0],0,0,0]];
ENDMODULE

